{attribute wpf [Container(Layout.Wrap)]}
{attribute wpf [Group(Layout.GroupBox)]}
FUNCTION_BLOCK fbPneumaticActuator
VAR_INPUT
	{attribute wpf [Container(Layout.Stack)]}
	{attribute clr [ReadOnly()]}
	{attribute addProperty Name "Retracted"}
	{attribute addProperty ToolTip "Sensor indicating that the actuator is retracted"}
	inRetracted : BOOL;
	{attribute clr [ReadOnly()]}
	{attribute addProperty Name "Extended"}
	{attribute addProperty ToolTip "Sensor indicating that the actuator is extended"}
	inExtended : BOOL;
END_VAR
VAR_OUTPUT
	{attribute wpf [Container(Layout.Stack)]}
	{attribute clr [ReadOnly()]}
	{attribute addProperty Name "Retract"}
	{attribute addProperty ToolTip "Signal for retracting"}
	outRetract : BOOL;
	{attribute clr [ReadOnly()]}
	{attribute addProperty Name "Extend"}
	{attribute addProperty ToolTip "Signal for extending"}
	outExtend : BOOL;
END_VAR
VAR
	{attribute wpf [Container(Layout.Stack)]}
	{attribute addProperty Name "Manual Retract"}
	{attribute addProperty ToolTip "Executes retraction in manual mode"}
	_manualRetract : BOOL;
	{attribute addProperty Name "Manual Extend"}
	{attribute addProperty ToolTip "Executes extension in manual mode"}
	_manualExtend : BOOL;
	{attribute 'hide'}
	_simulatedPosition : INT;
END_VAR

METHOD Extend : BOOL
VAR_INPUT
END_VAR
THIS^.outRetract := FALSE;
THIS^.outExtend := TRUE;

Extend := THIS^.inExtended;
END_METHOD

METHOD Manual : BOOL
VAR_INPUT
END_VAR
IF(THIS^._manualExtend AND_THEN THIS^.Extend()) THEN THIS^._manualExtend := FALSE; END_IF;
IF(THIS^._manualRetract AND_THEN THIS^.Retract()) THEN THIS^._manualRetract := FALSE; END_IF;

THIS^._manualExtend := FALSE;
THIS^._manualRetract := FALSE;
END_METHOD

METHOD Retract : BOOL
VAR_INPUT
END_VAR
THIS^.outRetract := TRUE;
THIS^.outExtend := FALSE;

Retract := THIS^.inRetracted;
END_METHOD

METHOD SimulateInputs : BOOL
VAR_INPUT
END_VAR
IF THIS^.outExtend THEN
	THIS^.inRetracted := FALSE;
	_simulatedPosition := _simulatedPosition + 1;
	IF _simulatedPosition >= 100 THEN
		_simulatedPosition := 100;
		THIS^.inExtended := TRUE;
	END_IF
END_IF
IF outRetract THEN
	THIS^.inExtended := FALSE;
	_simulatedPosition := _simulatedPosition - 1;
	IF _simulatedPosition <= -100 THEN
		_simulatedPosition := -100;
		THIS^.inRetracted := TRUE;
	END_IF
END_IF
END_METHOD

END_FUNCTION_BLOCK

(* stored: Version 1.1.0.1, ProductVersion 3.1.4024.2
   POU fbPneumaticActuator: Id {62afcfcf-c61c-4ad2-9fa1-449d45693563}, SpecialFunc None
   Method Extend: Id {178ca14c-8244-4ed4-b4ef-c91570455acf}
   Method Manual: Id {7d648aee-53bd-4128-8080-50b29e765f96}
   Method Retract: Id {a370ce29-ef9c-48c3-bfac-10eabf79b7c6}
   Method SimulateInputs: Id {4a2691fc-f991-4c45-9791-d15e2c6c0969} *)
